Staubli VAL3: CartesianTrajPt.pjx

--- CartesianTrajPt.pjx ---
Parameters version=s7.7.2 stackSize=5000 millimeterUnit=true
Program file=start.pgx
Program file=stop.pgx
Data file=CartesianTrajPt.dtx

--- CartesianTrajPt.dtx ---
public num nSeq
public num nPosition[3]
public num nOrientation[4]
public num nVelocity
public num nAcceleration
public num nBlendingRadius
public num nDuration
